PROGRAM MAIN
VAR
	st_current_state		:	FSM_states		:= FSM_states.state_init;
	
	fb_edgeDed_yellow		: 	fb_edgeDetector;
	fb_edgeDed_blue			:	fb_edgeDetector;
	
	b_array_code			:	ARRAY[0..3] OF BOOL		:=	[FALSE,TRUE,FALSE,TRUE];
	i_currentIndex			:	INT;
	t_correctCounter		:	TIME := T#0MS;
	
	i_wait_CodeChange		:	INT;
	
	
END_VAR

CASE st_current_state OF
	FSM_states.state_init:

		st_current_state	:=	FSM_states.state_close;
	FSM_states.state_close:
	
		GVL_IO.b_red_lamp	:=	FALSE;
		GVL_IO.b_green_lamp	:=	FALSE;
		i_currentIndex		:=	0;
		t_correctCounter	:=	T#0MS;
		i_wait_CodeChange	:=	0;
		
		st_current_state	:=	FSM_states.state_check;
			
	FSM_states.state_check:
		
		fb_edgeDed_blue(b_inputVal:=GVL_IO.b_blue_button);
		fb_edgeDed_yellow(b_inputVal:=GVL_IO.b_yellow_button);
		IF fb_edgeDed_blue.b_risingEdge THEN
			IF b_array_code[i_currentIndex]=FALSE THEN
				i_currentIndex		:=	i_currentIndex+1;
			ELSE
				st_current_state	:=	FSM_states.state_wrong;	
			END_IF
		ELSIF fb_edgeDed_yellow.b_risingEdge THEN
			IF b_array_code[i_currentIndex]=TRUE THEN
				i_currentIndex		:=	i_currentIndex+1;
			ELSE
				st_current_state	:=	FSM_states.state_wrong;	
			END_IF
		ELSIF fb_edgeDed_blue.b_doubleActivate THEN
			st_current_state	:=	FSM_states.state_Res;			
		END_IF
		
		IF i_currentIndex > 3 THEN
			st_current_state		:=	FSM_states.state_open;	
		END_IF
	FSM_states.state_Res:
		t_correctCounter	:=	t_correctCounter+GVL_const.T_CLOCK_CICLE;
		IF t_correctCounter=T#50MS THEN
			GVL_IO.b_green_lamp		:= NOT GVL_IO.b_green_lamp;
			GVL_IO.b_red_lamp		:= NOT GVL_IO.b_red_lamp;
		ELSIF t_correctCounter=T#100MS THEN
			GVL_IO.b_green_lamp		:= NOT GVL_IO.b_green_lamp;
			GVL_IO.b_red_lamp		:= NOT GVL_IO.b_red_lamp;
		ELSIF t_correctCounter=T#150MS THEN
			GVL_IO.b_green_lamp		:= NOT GVL_IO.b_green_lamp;
			GVL_IO.b_red_lamp		:= NOT GVL_IO.b_red_lamp;
		ELSIF t_correctCounter=T#200MS THEN
			GVL_IO.b_green_lamp		:= NOT GVL_IO.b_green_lamp;
			GVL_IO.b_red_lamp		:= NOT GVL_IO.b_red_lamp;
		ELSIF t_correctCounter=T#250MS THEN
			GVL_IO.b_green_lamp		:= NOT GVL_IO.b_green_lamp;
			GVL_IO.b_red_lamp		:= NOT GVL_IO.b_red_lamp;
		ELSIF t_correctCounter>T#300MS THEN
			st_current_state	:= FSM_states.state_init;
		END_IF
	
	FSM_states.state_wrong:
		
		IF t_correctCounter < GVL_const.T_LIGHT_DURATION THEN
			GVL_IO.b_red_lamp		:=	TRUE;
			t_correctCounter		:=	t_correctCounter + GVL_const.T_CLOCK_CICLE;
		ELSE
			st_current_state		:=	FSM_states.state_init;
		END_IF
	
	FSM_states.state_open:
		
		IF t_correctCounter < GVL_const.T_LIGHT_DURATION THEN
			GVL_IO.b_green_lamp		:=	TRUE;
			t_correctCounter		:=	t_correctCounter + GVL_const.T_CLOCK_CICLE;
		ELSE
			st_current_state		:=	FSM_states.state_init;
		END_IF
		
		
		IF GVL_IO.b_blue_button AND GVL_IO.b_yellow_button THEN
			st_current_state		:= FSM_states.state_goChange;
			i_currentIndex			:=0;
		END_IF
		
	FSM_states.state_goChange:
	
		fb_edgeDed_blue(b_inputVal			:=	GVL_IO.b_blue_button);
		fb_edgeDed_yellow(b_inputVal		:=	GVL_IO.b_yellow_button);
		
		IF fb_edgeDed_blue.b_fallingEdge OR fb_edgeDed_yellow.b_fallingEdge THEN
			i_wait_CodeChange				:=	i_wait_CodeChange+1;
		END_IF
		IF i_wait_CodeChange > 1 THEN
			st_current_state				:=	FSM_states.state_codChange;
		END_IF
		
		
	FSM_states.state_codChange:
		GVL_IO.b_green_lamp			:=	TRUE;
		GVL_IO.b_red_lamp			:=	TRUE;
		
		fb_edgeDed_blue(b_inputVal			:=GVL_IO.b_blue_button);
		fb_edgeDed_yellow(b_inputVal		:=GVL_IO.b_yellow_button);
		
		IF fb_edgeDed_blue.b_risingEdge THEN
			b_array_code[i_currentIndex]	:=	FALSE;
			i_currentIndex					:=	i_currentIndex+1;
		ELSIF fb_edgeDed_yellow.b_risingEdge THEN
			b_array_code[i_currentIndex]	:=	TRUE;
			i_currentIndex					:=	i_currentIndex+1;
		END_IF
		
		IF i_currentIndex > 3 THEN
			st_current_state				:=	FSM_states.state_init;
		END_IF
	
		
	
		
	
	
END_CASE

END_PROGRAM

(* stored: Version 1.1.0.1, ProductVersion 3.1.4022.12
   POU MAIN: Id {76f6e05a-fb6a-493b-b972-fc3e698e9984}, SpecialFunc None *)
